// TwinCAT 3 PLC project PlcLib
// ProgramVersion: 3.1.4023.0
// libraries:
//   Tc2_Standard, * (Beckhoff Automation GmbH)
//   Tc2_System, * (Beckhoff Automation GmbH)
//   Tc2_TcpIp, * (Beckhoff Automation GmbH)
//   Tc3_DynamicMemory, * (Beckhoff Automation GmbH)
//   Tc3_EventLogger, * (Beckhoff Automation GmbH)
//   Tc3_Module, * (Beckhoff Automation GmbH)
// project tree:
//   DUTs/ FB_Object.TcPOU, FB_ObjectExt.TcPOU, FB_SecondObject.TcPOU, FB_ThirdObject.TcPOU, ITF_Object.TcIO, ITF_ObjectExt.TcIO, Struct1.TcDUT
//   EventLoggerClass/ ITcMessage_Ext.TcIO, TcMessage_Ext.TcPOU
//   PlcAdsHandler/ ADSReadBasic.TcPOU
//   / PlcTask.TcTTO
//   POUs/ DynamicMemoryTesting.TcPOU, InterfaceTesting.TcPOU, MAIN.TcPOU
//   TCPIPHandler/ ITF_TcpIpBase.TcIO, TCPIP_Base.TcPOU
//   TCPIPHandler/Tasks/ ITask.TcIO, SocketCloseTask.TcPOU, SocketConnectTask.TcPOU, SocketRecieveTask.TcPOU, SocketSendTask.TcPOU

CONFIGURATION PlcLib
    RESOURCE PLC ON TwinCAT3
        TASK PlcTask(INTERVAL := T#10ms, PRIORITY := 20);
        PROGRAM MAIN WITH PlcTask : MAIN;
    END_RESOURCE
END_CONFIGURATION

// ---- DUTs/Struct1.TcDUT
{attribute 'enable_dynamic_creation'}
TYPE Struct1 :
STRUCT
	bIn : BOOL;
	iIn : INT;
END_STRUCT
END_TYPE

// ---- DUTs/ITF_Object.TcIO
INTERFACE ITF_Object EXTENDS __System.IQueryInterface

PROPERTY Index : int
GET
END_GET
SET
END_SET
END_PROPERTY

END_INTERFACE

// ---- DUTs/ITF_ObjectExt.TcIO
INTERFACE ITF_ObjectExt EXTENDS __System.IQueryInterface

METHOD AddSomeValues : int
VAR_INPUT
	x : INT;
	y : INT;
END_VAR
END_METHOD

END_INTERFACE

// ---- EventLoggerClass/ITcMessage_Ext.TcIO
INTERFACE ITcMessage_Ext

METHOD Send : BOOL
VAR_INPUT
	eventType : Tc3_EventLogger.TcEventEntry;
	args : STRING(255);
END_VAR
END_METHOD

END_INTERFACE

// ---- TCPIPHandler/ITF_TcpIpBase.TcIO
INTERFACE ITF_TcpIpBase

METHOD ConnectToRobot : BOOL
VAR_INPUT
END_VAR
END_METHOD

METHOD DisconnectFromRobot : BOOL
VAR_INPUT
END_VAR
END_METHOD

METHOD GetData : ARRAY[0..1439] OF byte
VAR_INPUT
END_VAR
END_METHOD

METHOD IsConnected : BOOL
VAR_INPUT
END_VAR
END_METHOD

PROPERTY RemoteServerIP : T_IPv4Addr
GET
END_GET
SET
END_SET
END_PROPERTY

PROPERTY RemoteServerPort : UDINT
GET
END_GET
SET
END_SET
END_PROPERTY

END_INTERFACE

// ---- TCPIPHandler/Tasks/ITask.TcIO
INTERFACE ITask

METHOD Abort : BOOL
VAR_INPUT
END_VAR
END_METHOD

PROPERTY Busy : bool
GET
END_GET
END_PROPERTY

PROPERTY Done : bool
GET
END_GET
END_PROPERTY

PROPERTY Error : bool
GET
END_GET
END_PROPERTY

END_INTERFACE

// ---- POUs/MAIN.TcPOU
PROGRAM MAIN
VAR
END_VAR

InterfaceTesting();
DynamicMemoryTesting();

END_PROGRAM

// ---- POUs/InterfaceTesting.TcPOU
PROGRAM InterfaceTesting
VAR
	fbParent : FB_Object(FALSE,1);
	fbChild : FB_ObjectExt(FALSE,2);
	fbSecond : FB_SecondObject;
	
	//Declaration interface assignment
	iParent : ITF_Object := fbParent;
	iChild : ITF_ObjectExt;
	
	//Declaration interface injected through constructor
	fbThird : FB_ThirdObject(ParentObject := fbParent);
	bCastResult : BOOL;
END_VAR

//Interface assignment in code
iChild := fbChild;

//Interface in property takes the parent interface
//passing child class here
fbSecond.ParentObject := fbChild;

//use method call to test cast
//child passed in using parent interface, need to cast to use child interface methods
bCastResult := fbSecond.AttemptCast();

END_PROGRAM

// ---- DUTs/FB_Object.TcPOU
{attribute 'enable_dynamic_creation'}
FUNCTION_BLOCK FB_Object IMPLEMENTS ITF_Object
VAR_INPUT
END_VAR
VAR_OUTPUT
END_VAR
VAR
END_VAR

METHOD FB_init : BOOL
VAR_INPUT
	bInitRetains : BOOL; // if TRUE, the retain variables are initialized (warm start / cold start)
	bInCopyCode : BOOL;  // if TRUE, the instance afterwards gets moved into the copy code (online change)
	IsEnabled : BOOL;
	Index : INT;
END_VAR
END_METHOD

PROPERTY Index : int
GET
END_GET
SET
END_SET
END_PROPERTY

PROPERTY IsEnabled : bool
GET
END_GET
SET
END_SET
END_PROPERTY

END_FUNCTION_BLOCK

// ---- DUTs/FB_ObjectExt.TcPOU
FUNCTION_BLOCK FB_ObjectExt EXTENDS FB_Object IMPLEMENTS ITF_ObjectExt
VAR_INPUT
END_VAR
VAR_OUTPUT
END_VAR
VAR
END_VAR

METHOD AddSomeValues : int
VAR_INPUT
	x : INT;
	y : INT;
END_VAR
AddSomeValues := x + y;
END_METHOD

END_FUNCTION_BLOCK

// ---- DUTs/FB_SecondObject.TcPOU
FUNCTION_BLOCK FB_SecondObject
VAR_INPUT
END_VAR
VAR_OUTPUT
END_VAR
VAR
	_parentObject : ITF_Object;
	hResult : INT;
END_VAR

METHOD AttemptCast : BOOL
VAR_INPUT
END_VAR
VAR
	itfChild : ITF_ObjectExt;
END_VAR
IF __QUERYINTERFACE(_parentObject,itfChild) THEN
	hResult := itfChild.AddSomeValues(2,2);
	AttemptCast := TRUE;
END_IF
END_METHOD

PROPERTY ParentObject : ITF_Object
GET
ParentObject := _parentObject;
END_GET
SET
_parentObject := ParentObject;
END_SET
END_PROPERTY

END_FUNCTION_BLOCK

// ---- DUTs/FB_ThirdObject.TcPOU
FUNCTION_BLOCK FB_ThirdObject
VAR_INPUT
END_VAR
VAR_OUTPUT
END_VAR
VAR
	_parentObject : ITF_Object;
END_VAR

METHOD FB_init : BOOL
VAR_INPUT
	bInitRetains : BOOL; // if TRUE, the retain variables are initialized (warm start / cold start)
	bInCopyCode : BOOL;  // if TRUE, the instance afterwards gets moved into the copy code (online change)
	ParentObject : ITF_Object;
END_VAR
_parentObject := ParentObject;
END_METHOD

END_FUNCTION_BLOCK

// ---- POUs/DynamicMemoryTesting.TcPOU
PROGRAM DynamicMemoryTesting
VAR
	/////////////First example///////////
	CreateBasicUserStructs	: BOOL := FALSE;
	CreatArrayOfUserStructs	: BOOL := FALSE;
	bDelete			: BOOL := FALSE;
	StaticArrayUserStructs 	: ARRAY [1..10] OF POINTER TO Struct1;
	DynamicArrayUserStructs	: POINTER TO POINTER TO Struct1;
	nIdx			: INT;
	nMax 			: INT := 10;

	///////////Second example//////////
	CreateBasicUserObjects: BOOL;
	CreateArrayUserObjects: BOOL;
	StaticArrayUserObjects 	: ARRAY [1..10] OF POINTER TO FB_Object;
	DymanicArrayUserObjects	: POINTER TO POINTER TO FB_Object;
	
	///////////Third Example////////////
	fbMem : Tc3_DynamicMemory.FB_DynMem_Manager2;
	ptrFbMem: POINTER TO Struct1;
	CreateBasicUserObject : bool;
	DeleteBasicUserObject: BOOL;
	CheckAllocatedMemory: BOOL;
	AllocatedMemory: ULINT;
END_VAR

////////////First Example - dynamic creation of user object/////////////////
IF CreateBasicUserStructs THEN
	FOR nIdx := 1 TO 10 DO
		StaticArrayUserStructs[nIdx] := __NEW(Struct1);
	END_FOR
	CreateBasicUserStructs := FALSE;
END_IF

IF CreatArrayOfUserStructs THEN
	DynamicArrayUserStructs := __NEW(POINTER TO Struct1, nMax);
	
	FOR nIdx := 0 TO nMax-1 DO
		DynamicArrayUserStructs[nIdx] := __NEW(Struct1);
	END_FOR

	CreatArrayOfUserStructs := FALSE;
END_IF

IF bDelete THEN
	__DELETE(DynamicArrayUserStructs);
	FOR nIdx := 1 TO 10 DO
		__DELETE(StaticArrayUserStructs[nIdx]);
	END_FOR
	bDelete := FALSE;
END_IF

///////////Second Example - dynamic creation of user object with parameter injection////////////////
IF CreateBasicUserObjects THEN
	FOR nIdx := 1 TO 10 DO
		StaticArrayUserObjects[nIdx] := __NEW(FB_Object(IsEnabled := TRUE, Index := 0));
	END_FOR
	CreateBasicUserObjects := FALSE;	
END_IF

IF CreateArrayUserObjects THEN
	DymanicArrayUserObjects := __NEW(POINTER TO FB_Object, nMax);
	
	FOR nIdx := 0 TO nMax-1 DO
		DymanicArrayUserObjects[nIdx] := __NEW(FB_Object(IsEnabled := TRUE, Index := nIdx));
	END_FOR
END_IF

IF bDelete THEN
	__DELETE(DymanicArrayUserObjects);
	FOR nIdx := 1 TO 10 DO
		__DELETE(StaticArrayUserObjects[nIdx]);
	END_FOR
	bDelete := FALSE;
END_IF

////////////Third Example - Dynamic creation using FB_DynMem class///////////////////
////////This is the new preferred method of dynamic memory allocation////////////
IF CreateBasicUserObject THEN
	ptrFbMem := fbMem.Alloc(nSize := SIZEOF(Struct1),bReset := TRUE);
	CreateBasicUserObject := FALSE;
END_IF

IF DeleteBasicUserObject THEN
	fbMem.Free2(ptrFbMem);
	DeleteBasicUserObject := FALSE;
END_IF

IF CheckAllocatedMemory THEN
	AllocatedMemory := fbMem.nAllocatedSize;
	CheckAllocatedMemory := FALSE;
END_IF

END_PROGRAM

// ---- EventLoggerClass/TcMessage_Ext.TcPOU
FUNCTION_BLOCK TcMessage_Ext IMPLEMENTS ITcMessage_Ext
VAR_INPUT
END_VAR
VAR_OUTPUT
END_VAR
VAR
    fbMsg : FB_TcMessage; 
	fbTest : Tc3_EventLogger.FB_TcEvent;
	fbInfo : Tc3_EventLogger.FB_TcSourceInfo;
	_loggerLevel : TcEventSeverity := TcEventSeverity.Info;
END_VAR

PROPERTY PUBLIC LoggerLevel : TcEventSeverity
GET
LoggerLevel := _loggerLevel;
END_GET
SET
_loggerLevel := LoggerLevel;
END_SET
END_PROPERTY

METHOD PUBLIC Send : BOOL
VAR_INPUT
	eventType : Tc3_EventLogger.TcEventEntry;
	args : STRING(255);
END_VAR
IF eventType.eSeverity >= LoggerLevel THEN
	THIS^.fbMsg.CreateEx(eventType, 0);
	THIS^.fbMsg.ipArguments.AddString(args);
	THIS^.fbMsg.Send(0);
	THIS^.fbMsg.Release();
END_IF
END_METHOD

END_FUNCTION_BLOCK

// ---- PlcAdsHandler/ADSReadBasic.TcPOU
FUNCTION_BLOCK ADSReadBasic
VAR_INPUT
END_VAR
VAR_OUTPUT
END_VAR
VAR
	AdsRead : ADSREAD;
	rtrig : R_TRIG;
	ReadState : INT;
	_Busy : BOOL;
	_done : BOOL;
END_VAR

//Sequence
CASE ReadState OF
	0://Wait for Read Command
		IF rtrig.Q THEN
			_done := FALSE;
			_Busy := TRUE;
			AdsRead.READ := TRUE;
			ReadState := 10;
		END_IF
	10://Wait for read busy
		IF AdsRead.BUSY THEN
			ReadState := 20;
		END_IF
	20://Wait for execute finish
		IF NOT AdsRead.BUSY THEN
			_Busy := FALSE;
			_done := true;
			AdsRead.READ := FALSE;
			rtrig.CLK := FALSE;
			ReadState := 0;
		END_IF
END_CASE

//Outputs

//FBs
rtrig();
AdsRead(TMOUT := T#5S);

PROPERTY Busy : BOOL
GET
Busy := THIS^._Busy;
END_GET
END_PROPERTY

PROPERTY Done : BOOL
GET
Done := _done;
END_GET
END_PROPERTY

{warning 'add property implementation'}
PROPERTY Error : BOOL
GET
Error := AdsRead.ERR;
END_GET
END_PROPERTY

{warning 'add property implementation'}
PROPERTY ErrorId : UDINT
GET
ErrorId := AdsRead.ERRID;
END_GET
END_PROPERTY

METHOD PUBLIC Execute : BOOL
VAR_INPUT
END_VAR
 IF NOT rtrig.CLK THEN
	 rtrig.CLK := true;
 END_IF
END_METHOD

METHOD PUBLIC SetADSReadTarget : BOOL
VAR_INPUT
	TargetNetId     : T_AmsNetId;
    TargetPort      : T_AmsPort;
    AdsIdxGrp    : UDINT;
    AdsIdxOff   : UDINT;
    ReadLength       : UDINT;
    ReadVarAddr  : PVOID;	
END_VAR
AdsRead.DESTADDR := ReadVarAddr;
AdsRead.IDXGRP := AdsIdxGrp;
AdsRead.IDXOFFS := AdsIdxOff;
AdsRead.LEN := ReadLength;
AdsRead.NETID := TargetNetId;
AdsRead.PORT := TargetPort;
END_METHOD

END_FUNCTION_BLOCK

// ---- TCPIPHandler/Tasks/SocketCloseTask.TcPOU
FUNCTION_BLOCK SocketCloseTask IMPLEMENTS ITask
VAR_INPUT
END_VAR
VAR_OUTPUT
END_VAR
VAR
	iState: INT;
	_done: BOOL;
	_busy: BOOL;
	_error: BOOL;
	_execute : BOOL;
	fbSocketClose : Tc2_TcpIp.FB_SocketClose;
END_VAR

CASE iState OF
	0:
		IF _execute THEN
			_done := FALSE;
			_busy := TRUE;
			_error := FALSE;
			fbSocketClose.bExecute := TRUE;
			IF fbSocketClose.bBusy THEN
				iState := 10;
				_execute := false;
			END_IF
		END_IF
	10:
		IF NOT fbSocketClose.bBusy THEN
			IF NOT fbSocketClose.bError THEN
				_done := TRUE;
			ELSE
				_error := TRUE;
			END_IF
			_busy := FALSE;
			fbSocketClose.bExecute := FALSE;
			iState := 0;
		END_IF
END_CASE

fbSocketClose(tTimeout := Tc2_System.DEFAULT_ADS_TIMEOUT);

METHOD Abort : BOOL
fbSocketClose.bExecute := FALSE;
_busy := FALSE;
_execute := FALSE;
Abort := TRUE;
iState := 0;
END_METHOD

PROPERTY Busy : BOOL
GET
Busy := _busy;
END_GET
END_PROPERTY

PROPERTY Done : BOOL
GET
Done := _done;
END_GET
END_PROPERTY

PROPERTY Error : BOOL
GET
Error := _error;
END_GET
END_PROPERTY

METHOD Execute : BOOL
VAR_INPUT
	remoteSocket: T_HSOCKET;
END_VAR
IF NOT fbSocketClose.bBusy THEN
	fbSocketClose.hSocket := remoteSocket;
	Execute := _execute := true;
END_IF
END_METHOD

END_FUNCTION_BLOCK

// ---- TCPIPHandler/Tasks/SocketConnectTask.TcPOU
FUNCTION_BLOCK SocketConnectTask IMPLEMENTS ITask
VAR_INPUT
END_VAR
VAR_OUTPUT
END_VAR
VAR
	_execute : BOOL;
	iState: INT;
	_done: BOOL;
	_busy: BOOL;
	_error: BOOL;
	fbSocketConnect : Tc2_TcpIp.FB_SocketConnect;
END_VAR

CASE iState OF
	0:
		IF _execute THEN
			_done := FALSE;
			_busy := TRUE;
			_error := FALSE;
			fbSocketConnect.bExecute := TRUE;
			IF fbSocketConnect.bBusy THEN
				iState := 10;
				_execute := false;
			END_IF
		END_IF
	10:
		IF NOT fbSocketConnect.bBusy THEN
			IF NOT fbSocketConnect.bError THEN
				_done := TRUE;
			ELSE
				_error := TRUE;
			END_IF
			_busy := FALSE;
			fbSocketConnect.bExecute := FALSE;
			iState := 0;
		END_IF
END_CASE

fbSocketConnect(tTimeout := Tc2_System.DEFAULT_ADS_TIMEOUT);

METHOD Abort : BOOL
fbSocketConnect.bExecute := FALSE;
_busy := FALSE;
_execute := FALSE;
Abort := TRUE;
iState := 0;
END_METHOD

PROPERTY Busy : BOOL
GET
Busy := _busy;
END_GET
END_PROPERTY

PROPERTY Done : BOOL
GET
Done := _done;
END_GET
END_PROPERTY

PROPERTY Error : BOOL
GET
Error := _error;
END_GET
END_PROPERTY

METHOD Execute : BOOL
VAR_INPUT
	RemoteIPAddress : Tc2_System.T_IPv4Addr;
	RemotePortNumber : UDINT;
END_VAR
IF NOT fbSocketConnect.bBusy THEN
	fbSocketConnect.sRemoteHost := RemoteIPAddress;
	fbSocketConnect.nRemotePort := RemotePortNumber;	
	Execute := _execute := TRUE;
END_IF
END_METHOD

PROPERTY PUBLIC RemoteSocket : T_HSOCKET
GET
RemoteSocket := fbSocketConnect.hSocket;
END_GET
END_PROPERTY

END_FUNCTION_BLOCK

// ---- TCPIPHandler/Tasks/SocketRecieveTask.TcPOU
FUNCTION_BLOCK SocketRecieveTask IMPLEMENTS ITask
VAR_INPUT
END_VAR
VAR_OUTPUT
	rxBuffer : ARRAY[0..1439] OF BYTE;
END_VAR
VAR
	iState: INT;
	_done: BOOL;
	_busy: BOOL;
	_error: BOOL;
	_execute: BOOL;
	fbSocketRecieve : Tc2_TcpIp.FB_SocketReceive;
	
	fbReceiveTimer : Tc2_Standard.TON;
END_VAR

CASE iState OF
	0:
		IF _execute THEN
			_done := FALSE;
			_busy := TRUE;
			_error := FALSE;
			iState := 5;
			_execute := FALSE;
		END_IF
		
	5:	
		fbReceiveTimer.IN := TRUE;
		fbSocketRecieve.bExecute := TRUE;
		IF fbReceiveTimer.Q THEN
			iState := 10;
			fbReceiveTimer.IN := FALSE;
		END_IF
	10:
		fbSocketRecieve.bExecute := FALSE;
		IF NOT fbSocketRecieve.bBusy THEN
			IF NOT fbSocketRecieve.bError THEN
				IF (fbSocketRecieve.nRecBytes > 0) THEN
					_busy := FALSE;
					_done := TRUE;
					iState := 0;
				ELSE
					iState := 5;
				END_IF
			ELSE
				_error := TRUE;
				_busy := FALSE;
				fbSocketRecieve.bExecute := FALSE;
				iState := 0;
			END_IF
			
		END_IF
END_CASE
fbReceiveTimer(PT := T#100MS);
fbSocketRecieve(pDest := ADR(rxBuffer),
				cbLen := SIZEOF(rxBuffer),
				tTimeout := Tc2_System.DEFAULT_ADS_TIMEOUT);

METHOD Abort : BOOL
fbSocketRecieve.bExecute := FALSE;
_busy := FALSE;
_execute := FALSE;
Abort := TRUE;
iState := 0;
END_METHOD

PROPERTY Busy : BOOL
GET
Busy := _busy;
END_GET
END_PROPERTY

PROPERTY Done : BOOL
GET
Done := _done;
END_GET
END_PROPERTY

PROPERTY Error : BOOL
GET
Error := _error;
END_GET
END_PROPERTY

METHOD Execute : BOOL
IF NOT fbSocketRecieve.bBusy THEN
	Execute := _execute := true;
END_IF
END_METHOD

PROPERTY PUBLIC RemoteSocket : T_HSOCKET
GET // PUBLIC
RemoteSocket := fbSocketRecieve.hSocket;
END_GET
SET // PUBLIC
fbSocketRecieve.hSocket := RemoteSocket;
END_SET
END_PROPERTY

END_FUNCTION_BLOCK

// ---- TCPIPHandler/Tasks/SocketSendTask.TcPOU
FUNCTION_BLOCK SocketSendTask IMPLEMENTS ITask
VAR_INPUT
END_VAR
VAR_OUTPUT
END_VAR
VAR
	iState: INT;
	_done: BOOL;
	_busy: BOOL;
	_error: BOOL;
	_execute : BOOL;
	fbSocketSend : Tc2_TcpIp.FB_SocketSend;
END_VAR

CASE iState OF
	0:
		IF _execute THEN
			_done := FALSE;
			_busy := TRUE;
			_error := FALSE;
			fbSocketSend.bExecute := TRUE;
			IF fbSocketSend.bBusy THEN
				iState := 10;
				_execute := false;
			END_IF
		END_IF
	10:
		IF NOT fbSocketSend.bBusy THEN
			IF NOT fbSocketSend.bError THEN
				_done := TRUE;
			ELSE
				_error := TRUE;
			END_IF
			_busy := FALSE;
			fbSocketSend.bExecute := FALSE;
			iState := 0;
		END_IF
END_CASE

fbSocketSend(tTimeout := Tc2_System.DEFAULT_ADS_TIMEOUT);

METHOD Abort : BOOL
fbSocketSend.bExecute := FALSE;
_busy := FALSE;
_execute := FALSE;
Abort := TRUE;
iState := 0;
END_METHOD

PROPERTY Busy : BOOL
GET
Busy := _busy;
END_GET
END_PROPERTY

PROPERTY Done : BOOL
GET
Done := _done;
END_GET
END_PROPERTY

PROPERTY Error : BOOL
GET
Error := _error;
END_GET
END_PROPERTY

METHOD Execute : BOOL
VAR_INPUT
	DataToSend : POINTER TO BYTE;
	DataLength : UDINT;
END_VAR
IF NOT fbSocketSend.bBusy THEN
	fbSocketSend.pSrc := DataToSend;
	fbSocketSend.cbLen := DataLength;
	Execute := _execute := true;
END_IF
END_METHOD

PROPERTY PUBLIC RemoteSocket : T_HSOCKET
GET // PUBLIC
RemoteSocket := fbSocketSend.hSocket;
END_GET
SET // PUBLIC
fbSocketSend.hSocket := RemoteSocket;
END_SET
END_PROPERTY

END_FUNCTION_BLOCK

// ---- TCPIPHandler/TCPIP_Base.TcPOU
FUNCTION_BLOCK TCPIP_Base IMPLEMENTS ITF_TcpIpBase
VAR_INPUT
END_VAR
VAR_OUTPUT
END_VAR
VAR
	connectToServer : SocketConnectTask;
	closeConectionToServer : SocketCloseTask;
	getReceivedDataFromServer : SocketRecieveTask;
	sendDataToServer : SocketSendTask;
	iState : INT;
	_connect: BOOL;
	_remoteIP : T_IPv4Addr;
	_remotePort : UDINT;
	_remoteHandle : Tc2_TcpIp.T_HSOCKET;
	clearRecieve: BOOL;
	_disconnect: BOOL;
	_connected: BOOL;
END_VAR

CASE iState OF
	0: 
		IF _connect THEN
			_connect := false;
			iState := 10;
		END_IF
		
	10:
		IF connectToServer.Execute(RemoteIPAddress := _remoteIP, 
									RemotePortNumber := _remotePort) THEN
			iState := 20;
		END_IF
		
	20:
		_remoteHandle := connectToServer.RemoteSocket;
		getReceivedDataFromServer.RemoteSocket := _remoteHandle;
		IF connectToServer.Done AND _remoteHandle.handle <> 0 THEN
			iState := 30;
			_connected := TRUE;
		END_IF
	
	30:
		IF getReceivedDataFromServer.Execute() THEN
			iState := 40;
		END_IF
		
	40:
		IF getReceivedDataFromServer.Done THEN
			IF _disconnect THEN
				_disconnect := FALSE;
				iState := 50;
			ELSE
				iState := 30;
			END_IF
			
		END_IF
	
	50:
		IF closeConectionToServer.Execute(remoteSocket := _remoteHandle) THEN
			iState := 60;
		END_IF
		
	60:
		IF closeConectionToServer.Done THEN
			iState := 0;
			_connected := FALSE;
		END_IF
		
			
END_CASE

connectToServer();
closeConectionToServer();
getReceivedDataFromServer();
sendDataToServer();

METHOD ConnectToRobot : BOOL
VAR_INPUT
END_VAR
ConnectToRobot := _connect := true;
END_METHOD

METHOD DisconnectFromRobot : BOOL
VAR_INPUT
END_VAR
DisconnectFromRobot := _disconnect := true;
END_METHOD

METHOD PUBLIC GetData : ARRAY[0..1439] OF byte
VAR_INPUT
END_VAR
GetData := getReceivedDataFromServer.rxBuffer;
END_METHOD

METHOD PUBLIC IsConnected : BOOL
VAR_INPUT
END_VAR
IsConnected := _connected;
END_METHOD

PROPERTY PUBLIC RemoteServerIP : T_IPv4Addr
GET
RemoteServerIP := _remoteIP;
END_GET
SET
_remoteIP := RemoteServerIP;
END_SET
END_PROPERTY

PROPERTY PUBLIC RemoteServerPort : udint
GET
RemoteServerPort := _remotePort;
END_GET
SET
_remotePort := RemoteServerPort;
END_SET
END_PROPERTY

END_FUNCTION_BLOCK
